INTERFACE INTERNAL I_StateInternal

METHOD INTERNAL _CanActivate : BOOL
VAR_INPUT
END_VAR
END_METHOD

METHOD INTERNAL _CanDeactivate : BOOL
VAR_INPUT
END_VAR
END_METHOD

PROPERTY INTERNAL _InQueue : BOOL
GET
END_GET
SET
END_SET
END_PROPERTY

PROPERTY INTERNAL _NextInBuffer : I_State
GET
END_GET
SET
END_SET
END_PROPERTY

METHOD INTERNAL _OnEntry
VAR_INPUT
END_VAR
END_METHOD

METHOD INTERNAL _OnExecute
VAR_INPUT
END_VAR
END_METHOD

METHOD INTERNAL _OnExit
VAR_INPUT
END_VAR
END_METHOD

(*
Returns the entity that owns this state.
*)
PROPERTY Owner : I_Entity
GET
END_GET
END_PROPERTY

END_INTERFACE

(* stored: Version 1.1.0.1
   Itf I_StateInternal: Id {b49468d8-74b2-4523-9a8e-300190600643}
   Folder _: Id {ea11d2f9-a8d0-4b23-897a-d4e88ba71fee}
   Folder Can: Id {6780bbc3-1843-4271-8203-ac0040ac9e3c}
   Folder On: Id {e8f03b0b-d8dc-462c-b1a1-c35c1e2a61ed}
   Method _CanActivate: Id {f8f7be64-9c99-4fdf-81b1-a2add969bdf5}
   Method _CanDeactivate: Id {ab838055-e4d5-46d5-a42d-ccdc9271d26a}
   Property _InQueue: Id {02ccade8-718f-4090-82d6-3da62d5eb7ab}
   Get Get: Id {5ec3504f-98d9-49cd-a289-f02c6221e357}
   Set Set: Id {4dc69405-ced6-4d6e-a2e0-c8d41c29999e}
   Property _NextInBuffer: Id {9d69fbbb-f40c-44f5-a73c-7b16ee2630e0}
   Get Get: Id {d75c9538-b75a-4f1f-96c4-0ffdef60e1b2}
   Set Set: Id {5569cd80-7757-474c-8eac-16d82fafea70}
   Method _OnEntry: Id {34f20feb-a6b8-476a-ac7d-107b73173ddd}
   Method _OnExecute: Id {23860f66-3827-4c1c-aa60-c228bf755ba9}
   Method _OnExit: Id {387ee35a-ce91-409e-90a2-90039f63ee69}
   Property Owner: Id {d93a7a3f-73d8-4f22-af14-97d5aa90489a}
   Get Get: Id {ada6f75c-eaf0-4d2e-ae8a-ddb0ab50f119} *)
